// TwinCAT 3 PLC project PLC
// ProgramVersion: 3.1.4023.0
// libraries:
//   Tc2_Standard, * (Beckhoff Automation GmbH)
//   Tc2_System, * (Beckhoff Automation GmbH)
//   Tc3_Module, * (Beckhoff Automation GmbH)
// project tree:
//   DUTs/ Command.TcDUT, State.TcDUT
//   / PlcTask.TcTTO
//   POUs/ Relay.TcPOU, Oven.TcPOU, MAIN.TcPOU, StateMachine.TcPOU

CONFIGURATION PLC
    RESOURCE PLC ON TwinCAT3
        TASK PlcTask(INTERVAL := T#10ms, PRIORITY := 20);
        PROGRAM MAIN WITH PlcTask : MAIN;
    END_RESOURCE
END_CONFIGURATION

// ---- DUTs/Command.TcDUT
{attribute 'qualified_only'}
{attribute 'strict'}
TYPE Command :
(
    Off := 0,
    On
);
END_TYPE

// ---- DUTs/State.TcDUT
{attribute 'qualified_only'}
{attribute 'strict'}
{attribute 'to_string'}
TYPE State :
(
    Off := 0,
    TurningOff,
    On,
    TurningOn
);
END_TYPE

// ---- POUs/MAIN.TcPOU
PROGRAM MAIN
VAR
    relay : Relay;
    oven : Oven;
END_VAR

// Oven command comes from the HMI
oven(relayState:=relay._state);
relay(_command:=oven.relayCommand);

END_PROGRAM

// ---- POUs/Relay.TcPOU
FUNCTION_BLOCK Relay EXTENDS StateMachine
VAR
    relayOnFeedback AT %I* : BOOL;
    turnOnRelay AT %Q* : BOOL;
END_VAR

SUPER^();

CASE _state OF
    State.Off :
        IF _command = Command.On THEN
            _state := State.TurningOn;
        END_IF
    State.TurningOn :
        turnOnRelay := TRUE;
        IF relayOnFeedback THEN
            _state := State.On;
        END_IF
        IF _command = Command.Off THEN
            _state := State.TurningOff;
        END_IF
    State.On :
        IF _command = Command.Off THEN
            _state := State.TurningOff;
        END_IF
    State.TurningOff :
        turnOnRelay := FALSE;
        IF NOT relayOnFeedback THEN
            _state := State.Off;
        END_IF
        IF _command = Command.On THEN
            _state := State.TurningOn;
        END_IF
END_CASE

END_FUNCTION_BLOCK

// ---- POUs/StateMachine.TcPOU
FUNCTION_BLOCK StateMachine
VAR_INPUT
    _command : Command;
END_VAR
VAR_OUTPUT
    _state : State;
END_VAR
VAR
    _stateName : STRING;
END_VAR

_stateName := TO_STRING(_state);

END_FUNCTION_BLOCK

// ---- POUs/Oven.TcPOU
FUNCTION_BLOCK Oven EXTENDS StateMachine
VAR_INPUT
    relayState : State;
    targetTemperature : REAL;
END_VAR
VAR_OUTPUT
    relayCommand : Command;
END_VAR
VAR
    thermoCouple_Celcius AT %I* : REAL;
    heaterCurrent_Ampere AT %Q* : REAL;
END_VAR

SUPER^();

CASE _state OF
    State.Off :
        IF _command = Command.On THEN
            _state := State.TurningOn;
        END_IF
    State.TurningOn :
        relayCommand := Command.On;
        IF relayState = State.On THEN
            _state := State.On;
        END_IF

        IF _command = Command.Off THEN
            _state := State.TurningOff;
        END_IF
    State.On :
        heaterCurrent_Ampere := SQRT(targetTemperature);

        IF _command = Command.Off THEN
            _state := State.TurningOff;
        END_IF
    State.TurningOff :
        heaterCurrent_Ampere := 0;
        relayCommand := Command.Off;
        IF relayState = State.Off THEN
            _state := State.Off;
        END_IF
END_CASE

END_FUNCTION_BLOCK
